PROGRAM MAIN
VAR
	name 	: STRING;
	number 	: INT;
	Intermidiate : STRING;
		
END_VAR

END_PROGRAM

(* stored: Version 1.1.0.1, ProductVersion 3.1.4024.12
   POU MAIN: Id {295b4b94-25c4-4e63-899f-50b130b5e294}, SpecialFunc None *)
